Yaskawa INFORM job: SKINCORN.JBI

/JOB
//NAME SKINCORN
//POS
///NPOS 4,0,0,0,0,0
///TOOL 0
///POSTYPE PULSE
///PULSE
C00000=-35562,61890,18115,4528,-46926,14557
C00001=-2141,105169,80140,173,-71106,945
C00002=78912,55415,19027,-9564,-51017,-32636
C00003=70459,3614,-49719,-9391,-26268,-27780
//INST
///ATTR SC,RW
///GROUP1 RB1
NOP
MOVJ C00000 VJ=0.50
MOVJ C00001 VJ=0.50
MOVJ C00002 VJ=0.50
MOVJ C00003 VJ=0.50
MOVJ C00000 VJ=0.50
END
